// TIA Portal V20 export
TYPE "LKinCtrl_typePnPConveyorTracking"
   STRUCT
      enable : Bool;   // = TRUE: Set tracking with command execution
      conveyorBeltAxis : DB_ANY;   // Conveyor belt axis DB
      conveyorBeltOrigin : TO_Struct_Kinematics_Frame;   // Frame to origin of conveyor belt
      initialObjectPosition : TO_Struct_Kinematics_Frame;   // Initial object position on conveyor (only x allowed)
   END_STRUCT;
END_TYPE
